FUNCTION_BLOCK F_MAX (* maximum *)
  PACKAGE iec61131::selection;
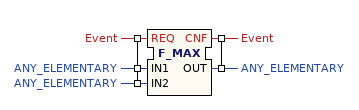
  EVENT_INPUT
    REQ WITH IN1, IN2; (* Service Request *)
  END_EVENT
  EVENT_OUTPUT
    CNF WITH OUT; (* Confirmation of Requested Service *)
  END_EVENT
  VAR_INPUT
    IN1 : ANY_ELEMENTARY; (* Input value 1 *)
    IN2 : ANY_ELEMENTARY; (* Input value 2 *)
  END_VAR
  VAR_OUTPUT
    OUT : ANY_ELEMENTARY; (* maximum value *)
  END_VAR
END_FUNCTION_BLOCK
